FUNCTION_BLOCK Crane_MoveToLSC EXTENDS Crane_MoveBase
VAR_INPUT
END_VAR
VAR_OUTPUT
END_VAR
VAR
	// (EProcessVariables.Crane_CylinderRetracted = TRUE) AND ((EProcessVariables.Crane_HoldingWorkpiece = FALSE) OR ((EProcessVariables.LSC_ProductType = 0) AND ((EProcessVariables.RFC_ProductType_1 = 0) AND (EProcessVariables.RFC_ProductType_2 = 0))))
	m_compExpr1: ComparisonExpression(EProcessVariables.Crane_CylinderRetracted, EComparisonType.equals, EDataType.binary, TRUE, 0, '', TRUE);
	m_compExpr3: ComparisonExpression(EProcessVariables.Crane_HoldingWorkpiece, EComparisonType.equals, EDataType.binary, FALSE, 0, '', TRUE);
	m_compExpr5: ComparisonExpression(EProcessVariables.LSC_ProductType, EComparisonType.equals, EDataType.numeric, FALSE, 0, '', TRUE);
	m_compExpr7: ComparisonExpression(EProcessVariables.RFC_ProductType_1, EComparisonType.equals, EDataType.numeric, FALSE, 0, '', TRUE);
	m_compExpr9: ComparisonExpression(EProcessVariables.RFC_ProductType_2, EComparisonType.equals, EDataType.numeric, FALSE, 0, '', TRUE);
	m_boolExpr10: BoolExpression(m_compExpr7, EBoolOperation.and_op, m_compExpr9);
	m_boolExpr11: BoolExpression(m_compExpr5, EBoolOperation.and_op, m_boolExpr10);
	m_boolExpr12: BoolExpression(m_compExpr3, EBoolOperation.or_op, m_boolExpr11);
	m_precondition: BoolExpression(m_compExpr1, EBoolOperation.and_op, m_boolExpr12);
	
	// EProcessVariables.Crane_AtLSC = TRUE
	m_postcondition: ComparisonExpression(EProcessVariables.Crane_AtLSC, EComparisonType.equals, EDataType.binary, TRUE, 0, '', TRUE);
END_VAR

SUPER^();

METHOD AtTarget : BOOL
VAR_INPUT
END_VAR
AtTarget := m_ptrCrane^.AtConveyor;
END_METHOD

METHOD FB_init : BOOL
VAR_INPUT
	bInitRetains : BOOL; // if TRUE, the retain variables are initialized (warm start / cold start)
	bInCopyCode : BOOL;  // if TRUE, the instance afterwards gets moved into the copy code (online change)
		
	i_ptrCrane: POINTER TO Crane;
END_VAR
m_ptrCrane := i_ptrCrane;

m_id := EPrimitives.Crane_MoveToLSC;
m_timeout := T#30S;

Precondition := m_precondition;
Postcondition := m_postcondition;

m_initDirection := TRUE;	//TRUE: Clockwise
m_targetTimeout := T#10S;
END_METHOD

END_FUNCTION_BLOCK

(* stored: Version 1.1.0.1, ProductVersion 3.1.4024.9
   POU Crane_MoveToLSC: Id {15eba410-d45b-4017-b72a-4a195c431512}, SpecialFunc None
   Method AtTarget: Id {b47b7b48-b787-416e-b0a5-337e3fb3b22b}
   Method FB_init: Id {cce78632-047d-49e3-ae7c-01dc75ff6324} *)
